SUBAPPLICATION SubApp_PC_B (* Geraet B (Station 12, 192.168.1.12): wie Training_11, aber Transport-Layer UND die Bridge/Interlock-Kette bleiben A2X-gebuendelt bis unmittelbar vor der physischen Hardware. EIN A2X2_CLIENT_2_0_SUBSCRIBE_2_PLUG uebernimmt den kompletten Roundtrip fuer UP+DOWN. MyLib::sys::A2X2_ILOCK_SWITCH_PROTECT kapselt Bridge (A2X2_TO_A2X), Interlock (ILOCK_SWITCH_PROTECT_A2X) und Split (A2X_SPLIT_2) in einem Composite (DT_PROTECT als Parameter) und liefert direkt den interlocked Zustand als A2X-Plug. MyLib::sys::A2X_TO_QXA2 kapselt - analog zu Softkey2_TO_A2X2_BG auf PC_A - das Entbuendeln auf die 2 physischen logiBUS_QXA-Ausgaenge. *)
  (* Standard: 61499-2; Description: Copyright (c) 2026 Meisterschulen am Ostbahnhof This program and the accompanying materials are made available under the terms of the Eclipse Public License 2.0 which is available at https://www.eclipse.org/legal/epl-2.0/ SPDX-License-Identifier: EPL-2.0 *)
  (* Version 1.0, 2026-09-05, Franz Höpfinger, Meisterschulen am Ostbahnhof, initial API and implementation and/or initial documentation *)
  PACKAGE subapp::Training_12_OPC_UA_RES;
  IMPORT VV::const::OPC_UA::myOpcUaAddresses::SW2_PRESS_LOCAL_READ;
  IMPORT VV::const::OPC_UA::myOpcUaAddresses::SW2_STATE_REMOTE_WRITE;
  IMPORT logiBUS::io::DQ::logiBUS_DO::Output_Q7;
  IMPORT logiBUS::io::DQ::logiBUS_DO::Output_Q8;
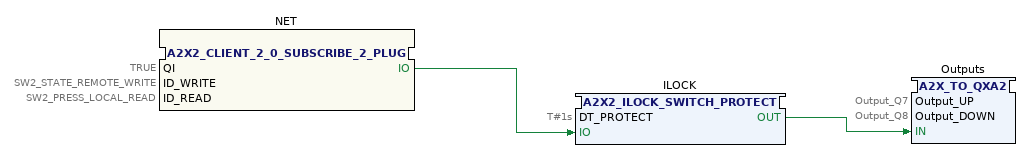
  FBS
    NET : adapter::net::A2X2_CLIENT_2_0_SUBSCRIBE_2_PLUG(QI := TRUE, ID_WRITE := SW2_STATE_REMOTE_WRITE, ID_READ := SW2_PRESS_LOCAL_READ);
  END_FBS
  SUBAPPS
    ILOCK : MyLib::sys::A2X2_ILOCK_SWITCH_PROTECT(DT_PROTECT := T#1s);
    Outputs : MyLib::sys::A2X_TO_QXA2(Output_UP := Output_Q7, Output_DOWN := Output_Q8);
  END_SUBAPPS
  ADAPTER_CONNECTIONS
    NET.IO TO ILOCK.IO;
    ILOCK.OUT TO Outputs.IN;
  END_CONNECTIONS
END_SUBAPPLICATION
